FUNCTION_BLOCK FB_LogWarningEdge
VAR_INPUT
   Event : BOOL; // Event flag
   Message : T_MaxString; // Log message
   EventFallingEdge : BOOL := FALSE; // Defined which edge: FALSE = rising TRUE = falling, 
END_VAR
VAR_OUTPUT
   Q : BOOL;
END_VAR
VAR
   fbLogEdge : FB_LogOnEdge;
END_VAR

fbLogEdge(
   Event := Event,
   Message := Message,
   LogSeverity := E_LogSeverity.Warning,
   EventFallingEdge := EventFallingEdge,
   Q => Q
);

END_FUNCTION_BLOCK

(* stored: Version 1.1.0.1, ProductVersion 3.1.4024.9
   POU FB_LogWarningEdge: Id {07beed0b-ff58-4e01-8d1d-4927c88129bb}, SpecialFunc None *)
